TYPE TPhaseDraining :
STRUCT
	Cmd : TPhaseCmd;
	State : TPhaseState;
	
	ParamDrainLevel : REAL;
	WaterLevel : REAL;
END_STRUCT
END_TYPE

(* stored: Version 1.1.0.1, ProductVersion 3.1.4024.12
   DUT TPhaseDraining: Id {32c7465a-c6e6-458f-ba2a-5e00c7fb7eef} *)
